INTERFACE I_AxisBase

END_INTERFACE

(* stored: Version 1.1.0.1
   Itf I_AxisBase: Id {0aa9fe18-9b82-4dd1-a575-8312f33b257a} *)
